VAR_GLOBAL
    Axis1 : AXIS_REF;
    Axis2 : AXIS_REF;
    Axis3 : AXIS_REF;
    Axis4 : AXIS_REF;
    Axis5 : AXIS_REF;
    Axis6 : AXIS_REF;
END_VAR

(* stored: Version 1.1.0.1, ProductVersion 3.1.4024.15
   GVL GVL_Axes: Id {053db407-795a-4050-8b69-23a92dc2826b} *)
